PROGRAM MAIN
VAR
	main_fsm	: Main_FSM;
	main_tests	: FB_Test_FSM;
	
	tests_on	: BOOL	:= TRUE;
END_VAR

IF tests_on THEN
	TcUnit.RUN();
ELSE
	main_fsm();
END_IF

END_PROGRAM

(* stored: Version 1.1.0.1
   POU MAIN: Id {ee0ed416-3c8e-41d0-b63e-3e0aab4b08ba}, SpecialFunc None *)
